{attribute 'no_check'}
//Provides the countdown value of an TON timer
FUNCTION getTonCountdown : TIME
VAR_IN_OUT
	Timer													:	TON;
END_VAR
VAR
END_VAR

IF Timer.IN
	AND NOT Timer.Q
THEN
	getTonCountdown 										:= Timer.PT - Timer.ET;
ELSE
	getTonCountdown 										:= T#0MS;
END_IF

END_FUNCTION

(* stored: Version 1.1.0.1, ProductVersion 3.1.4024.3
   POU getTonCountdown: Id {263ca799-eba4-4078-a555-9d8d6c3d76e4}, SpecialFunc None *)
